FUNCTION_BLOCK PUBLIC FileExtensionNotSupportedError EXTENDS Error
VAR
	state : (CLEARED, RAISED);
	fileExtension : T_MAXSTRING;
END_VAR

PROPERTY Active : BOOL
GET
Active := state <> CLEARED;
END_GET
END_PROPERTY

METHOD PUBLIC Clear
fileExtension := '';
state := CLEARED;
END_METHOD

PROPERTY PUBLIC ErrorCode : HRESULT
GET
ErrorCode := Tc2_System.E_HRESULTAdsErr.ACCESSDENIED;
END_GET
END_PROPERTY

PROPERTY PUBLIC Message : T_MaxString
GET
Message := 'File Extension not supported';
END_GET
END_PROPERTY

METHOD PUBLIC Raise
VAR_INPUT
	FilePath : T_MAXSTRING;
END_VAR
VAR
	fileDrive : STRING(3);
    fileDirectory : T_MAXSTRING;
    fileName : T_MAXSTRING;
    fileExtension : T_MAXSTRING;
	graphSettings : I_GraphSettings;
END_VAR
F_SplitPathName(FilePath,fileDrive,fileDirectory,fileName,fileExtension);

THIS^.fileExtension := fileExtension;
state := RAISED;
END_METHOD

PROPERTY Reason : T_MAXSTRING
GET
Reason := fileExtension;
END_GET
END_PROPERTY

END_FUNCTION_BLOCK

(* stored: Version 1.1.0.1, ProductVersion 3.1.4024.12
   POU FileExtensionNotSupportedError: Id {7dd61429-883e-01af-2c51-0b664f08c11f}, SpecialFunc None
   Property Active: Id {4e99588a-4337-09d7-0b18-2c95a9c2af5f}
   Get Get: Id {a9106d0b-1b0e-0648-04ed-33dac9406f94}
   Method Clear: Id {8d45e83d-bc84-05da-1946-95ada49064b6}
   Property ErrorCode: Id {84efd0b1-b399-0229-3038-debc2c0abce3}
   Get Get: Id {b80607ef-3991-0275-05ab-e574a79a2eb8}
   Property Message: Id {9acabd2b-2469-0edb-2042-4d54c9e9ea58}
   Get Get: Id {bbe86dee-522b-0f13-225a-5dcc69ed6c83}
   Method Raise: Id {65f7b67c-786a-0cef-3d16-137888e19b05}
   Property Reason: Id {5c6ef694-2725-0c46-211b-c2ab49c71e56}
   Get Get: Id {6b8776c9-0426-05c7-3caa-e2930cff05ef} *)
